// TIA Portal V20 export
TYPE "RFID_BALLUFF_UDT"
   STRUCT
      Start : Bool;
      job_Type : Int;
      Adr_Recieve : Int;
      Adr_Send : Int;
      Addr_CodeTag : Int;
      Length_CodeTag : Int;
   END_STRUCT;
END_TYPE
